PROGRAM FB_RobotTCPListen
VAR_INPUT
	bEnable : BOOL;
	Robot : STRING;
END_VAR
VAR_OUTPUT
	bBusy : BOOL;
	bConnected : BOOL;
	bError : BOOL;
END_VAR
VAR
	eState : E_RobotTCPListen;
	StartTrigger : R_TRIG;
	StopTrigger : F_TRIG;
	
	fbSocketConnect : FB_SocketConnect := (sSrvNetId := '', tTimeout := DEFAULT_ADS_TIMEOUT);
	fbSocketClose : FB_SocketClose := (sSrvNetId := '', tTimeout := DEFAULT_ADS_TIMEOUT);
	fbSocketReceive : FB_SocketReceive := (sSrvNetId := '', tTimeout := DEFAULT_ADS_TIMEOUT, cbLen := 800);
	
	
	hSocket1: T_HSOCKET;
	
	data : ARRAY [0..800] OF BYTE;
	
END_VAR

// Execute interrupt checks
StartTrigger(CLK := bEnable);
StopTrigger(CLK := bEnable);

CASE eState OF
	eState.Idle:
		IF StartTrigger.Q THEN
			bBusy := TRUE;
			eState := eState.Connect_Start;
		ELSIF StopTrigger.Q THEN
			eState := eState.Close_Start;
		ELSIF bConnected THEN
			eState := eState.Receive_Start;
		END_IF
	
	eState.Connect_Start:
		fbSocketConnect.bExecute := TRUE;
		fbSocketConnect.nRemotePort := 30001;
		IF Robot='UR3' THEN
			fbSocketConnect.sRemoteHost := '192.168.1.3';
		ELSIF Robot='UR5' THEN
			fbSocketConnect.sRemoteHost := '192.168.1.5';
		ELSE
			eState := eState.HandleError;
		END_IF
		fbSocketConnect();
		eState := eState.Connect_Wait;
		
	eState.Connect_Wait:
		fbSocketConnect.bExecute := FALSE;	
		IF fbSocketConnect.bError THEN
			eState := eState.HandleError;
		ELSIF NOT fbSocketConnect.bBusy THEN
			bConnected := TRUE;
			hSocket1 := fbSocketConnect.hSocket;
			eState := eState.Idle;
		END_IF
		
	eState.Receive_Start:
		fbSocketReceive.bExecute := TRUE;
		fbSocketReceive.hSocket := hSocket1;
		fbSocketReceive.pDest := ADR(data);
		eState := eState.Receive_Wait;
	
	eState.Receive_Wait:
		fbSocketReceive.bExecute := FALSE;
		IF fbSocketReceive.bError THEN
			eState := eState.HandleError;
		ELSIF NOT fbSocketReceive.bBusy THEN
			eState := eState.Idle;
		END_IF
				
	eState.Close_Start:
		fbSocketClose.bExecute := TRUE;
		fbSocketClose.hSocket := hSocket1;
		eState := eState.Close_Wait;
	
	eState.Close_Wait:
		fbSocketClose.bExecute := FALSE;
		IF fbSocketClose.bError THEN
				eState := eState.HandleError;
		ELSIF NOT fbSocketClose.bBusy THEN
			bConnected := FALSE;
			MEMSET(ADR(hSocket1),0,SIZEOF(hSocket1));
			bBusy := FALSE;
			bError := FALSE;
			eState := eState.Idle;
		END_IF
		
	eState.HandleError:
		bError := TRUE;
		IF bConnected THEN
			eState := eState.Close_Start;
		ELSE
			bBusy := FALSE;
			eState := eState.Idle;
		END_IF
		
END_CASE

fbSocketConnect();
fbSocketReceive();
fbSocketClose();

END_PROGRAM

(* stored: Version 1.1.0.1, ProductVersion 3.1.4020.12
   POU FB_RobotTCPListen: Id {8049a8bc-c88a-46b6-885c-8d0914a443b2}, SpecialFunc None *)
